DATA_BLOCK "Pol_sklad_db"
{ S7_Optimized_Access := 'FALSE' }
VERSION : 0.1
   STRUCT
      Pol_p : Real;
      Eror_pol_p : DWord;
      S_pol : Real;
      Weigt : Real;
      Densyty : Real;
      "1_pol" : Struct
         Weight_db : Real;
         Weight_zero : Real;
         Weight_Formula_W_T : Real;
         Visible : Bool;
         p_zero : Real;
         p_weight : Real;
         Zero_but : Bool;
         Weight_but : Bool;
         S : Real;
         Densyty : Real;
         Korect : Bool;
      END_STRUCT;
      "2_pol" : Struct
         Weight_db : Real;
         Weight_zero : Real;
         Weight_Formula_W_T : Real;
         Visible : Bool;
         p_zero : Real;
         p_weight : Real;
         Zero_but : Bool;
         Weight_but : Bool;
         S : Real;
         Densyty : Real;
         Korect : Bool;
      END_STRUCT;
      "3_pol" : Struct
         Weight_db : Real;
         Weight_zero : Real;
         Weight_Formula_W_T : Real;
         Visible : Bool;
         p_zero : Real;
         p_weight : Real;
         Zero_but : Bool;
         Weight_but : Bool;
         S : Real;
         Densyty : Real;
         Korect : Bool;
      END_STRUCT;
      "4_pol" : Struct
         Weight_db : Real;
         Weight_zero : Real;
         Weight_Formula_W_T : Real;
         Visible : Bool;
         p_zero : Real;
         p_weight : Real;
         Zero_but : Bool;
         Weight_but : Bool;
         S : Real;
         Densyty : Real;
         Korect : Bool;
      END_STRUCT;
      "5_pol" : Struct
         Weight_db : Real;
         Weight_zero : Real;
         Weight_Formula_W_T : Real;
         Visible : Bool;
         p_zero : Real;
         p_weight : Real;
         Zero_but : Bool;
         Weight_but : Bool;
         S : Real;
         Densyty : Real;
         Korect : Bool;
      END_STRUCT;
      "6_pol" : Struct
         Weight_db : Real;
         Weight_zero : Real;
         Weight_Formula_W_T : Real;
         Visible : Bool;
         p_zero : Real;
         p_weight : Real;
         Zero_but : Bool;
         Weight_but : Bool;
         S : Real;
         Densyty : Real;
         Korect : Bool;
      END_STRUCT;
      "7_pol" : Struct
         Weight_db : Real;
         Weight_zero : Real;
         Weight_Formula_W_T : Real;
         Visible : Bool;
         p_zero : Real;
         p_weight : Real;
         Zero_but : Bool;
         Weight_but : Bool;
         S : Real;
         Densyty : Real;
         Korect : Bool;
      END_STRUCT;
      "8_pol" : Struct
         Weight_db : Real;
         Weight_zero : Real;
         Weight_Formula_W_T : Real;
         Visible : Bool;
         p_zero : Real;
         p_weight : Real;
         Zero_but : Bool;
         Weight_but : Bool;
         S : Real;
         Densyty : Real;
         Korect : Bool;
      END_STRUCT;
      "9_pol" : Struct
         Weight_db : Real;
         Weight_zero : Real;
         Weight_Formula_W_T : Real;
         Visible : Bool;
         p_zero : Real;
         p_weight : Real;
         Zero_but : Bool;
         Weight_but : Bool;
         S : Real;
         Densyty : Real;
         Korect : Bool;
      END_STRUCT;
      "10_pol" : Struct
         Weight_db : Real;
         Weight_zero : Real;
         Weight_Formula_W_T : Real;
         Visible : Bool;
         p_zero : Real;
         p_weight : Real;
         Zero_but : Bool;
         Weight_but : Bool;
         S : Real;
         Densyty : Real;
         Korect : Bool;
      END_STRUCT;
   END_STRUCT;


BEGIN
   Pol_p := 1.149812;
   Eror_pol_p := 16#0000_0000;
   S_pol := 6.819987;
   Weigt := 79.9358;
   Densyty := 1.35;
   "1_pol".Weight_db := 0.0;
   "1_pol".Weight_zero := 0.0;
   "1_pol".Weight_Formula_W_T := 81.81128;
   "1_pol".Visible := TRUE;
   "1_pol".p_zero := 0.0;
   "1_pol".p_weight := 0.0;
   "1_pol".Zero_but := FALSE;
   "1_pol".Weight_but := FALSE;
   "1_pol".S := 6.98;
   "1_pol".Densyty := 1.35;
   "1_pol".Korect := FALSE;
   "2_pol".Weight_db := 19.52373;
   "2_pol".Weight_zero := 0.0;
   "2_pol".Weight_Formula_W_T := 78.76387;
   "2_pol".Visible := FALSE;
   "2_pol".p_zero := 0.0;
   "2_pol".p_weight := 0.2850116;
   "2_pol".Zero_but := FALSE;
   "2_pol".Weight_but := FALSE;
   "2_pol".S := 6.72;
   "2_pol".Densyty := 1.35;
   "2_pol".Korect := FALSE;
   "3_pol".Weight_db := 0.0;
   "3_pol".Weight_zero := 0.0;
   "3_pol".Weight_Formula_W_T := 78.52945;
   "3_pol".Visible := FALSE;
   "3_pol".p_zero := 0.0;
   "3_pol".p_weight := 0.0;
   "3_pol".Zero_but := FALSE;
   "3_pol".Weight_but := FALSE;
   "3_pol".S := 6.7;
   "3_pol".Densyty := 1.35;
   "3_pol".Korect := FALSE;
   "4_pol".Weight_db := 73.68473;
   "4_pol".Weight_zero := 0.0;
   "4_pol".Weight_Formula_W_T := 78.76387;
   "4_pol".Visible := FALSE;
   "4_pol".p_zero := 0.0;
   "4_pol".p_weight := 1.075665;
   "4_pol".Zero_but := FALSE;
   "4_pol".Weight_but := FALSE;
   "4_pol".S := 6.72;
   "4_pol".Densyty := 1.35;
   "4_pol".Korect := FALSE;
   "5_pol".Weight_db := 24.61529;
   "5_pol".Weight_zero := 0.0;
   "5_pol".Weight_Formula_W_T := 77.55404;
   "5_pol".Visible := FALSE;
   "5_pol".p_zero := 0.0;
   "5_pol".p_weight := 0.364945;
   "5_pol".Zero_but := FALSE;
   "5_pol".Weight_but := FALSE;
   "5_pol".S := 6.61678;
   "5_pol".Densyty := 1.35;
   "5_pol".Korect := FALSE;
   "6_pol".Weight_db := 49.182;
   "6_pol".Weight_zero := 0.0;
   "6_pol".Weight_Formula_W_T := 78.64666;
   "6_pol".Visible := FALSE;
   "6_pol".p_zero := 0.0;
   "6_pol".p_weight := 0.7190394;
   "6_pol".Zero_but := FALSE;
   "6_pol".Weight_but := FALSE;
   "6_pol".S := 6.71;
   "6_pol".Densyty := 1.35;
   "6_pol".Korect := FALSE;
   "7_pol".Weight_db := 123.4003;
   "7_pol".Weight_zero := 0.0;
   "7_pol".Weight_Formula_W_T := 78.64666;
   "7_pol".Visible := FALSE;
   "7_pol".p_zero := 0.0;
   "7_pol".p_weight := 1.804109;
   "7_pol".Zero_but := FALSE;
   "7_pol".Weight_but := FALSE;
   "7_pol".S := 6.71;
   "7_pol".Densyty := 1.35;
   "7_pol".Korect := FALSE;
   "8_pol".Weight_db := -0.2724785;
   "8_pol".Weight_zero := 0.4211032;
   "8_pol".Weight_Formula_W_T := 78.74628;
   "8_pol".Visible := FALSE;
   "8_pol".p_zero := 0.006148727;
   "8_pol".p_weight := 0.002170139;
   "8_pol".Zero_but := FALSE;
   "8_pol".Weight_but := FALSE;
   "8_pol".S := 6.7185;
   "8_pol".Densyty := 1.35;
   "8_pol".Korect := FALSE;
   "9_pol".Weight_db := 126.8467;
   "9_pol".Weight_zero := 0.0;
   "9_pol".Weight_Formula_W_T := 78.97484;
   "9_pol".Visible := FALSE;
   "9_pol".p_zero := 0.0;
   "9_pol".p_weight := 1.846788;
   "9_pol".Zero_but := FALSE;
   "9_pol".Weight_but := FALSE;
   "9_pol".S := 6.738;
   "9_pol".Densyty := 1.35;
   "9_pol".Korect := FALSE;
   "10_pol".Weight_db := 27.88432;
   "10_pol".Weight_zero := 0.0;
   "10_pol".Weight_Formula_W_T := 77.55404;
   "10_pol".Visible := TRUE;
   "10_pol".p_zero := 0.0;
   "10_pol".p_weight := 0.4134114;
   "10_pol".Zero_but := FALSE;
   "10_pol".Weight_but := FALSE;
   "10_pol".S := 6.61678;
   "10_pol".Densyty := 1.35;
   "10_pol".Korect := FALSE;

END_DATA_BLOCK

